{attribute 'GeneratedUsingTerminal: AX8108-0100-0101-0101'}
{attribute addProperty BoxType "AX8108-0100-0101-0101"}
{attribute addProperty Id "Ch_A_ControlwordAT %Q*UINT2"}
{attribute addProperty CRC "2845499694"}
{attribute addProperty Size "2"}
TYPE Ch_A_AxisMain_Outputs_A99AE12E :
STRUCT
	{attribute addProperty Name "Ch_A_Controlword"}
	Ch_A_Controlword AT %Q* : UINT;
END_STRUCT
END_TYPE

(* stored: Version 1.2.0.0, ProductVersion 3.1.4024.9
   DUT Ch_A_AxisMain_Outputs_A99AE12E: Id {8b3c4679-ab82-4724-a239-825798a6d4fd} *)
